INTERFACE I_RpcApi

METHOD CyclicCall
VAR_INPUT
END_VAR
END_METHOD

METHOD RegisterAsynchronousRpcHandlersWith
VAR_INPUT
	Host : I_HostAsynchronousRpcHandlers;
END_VAR
END_METHOD

METHOD RegisterSynchronousRpcHandlersWith
VAR_INPUT
	Host : I_HostSynchronousRpcHandlers;
END_VAR
END_METHOD

END_INTERFACE

(* stored: Version 1.1.0.1, ProductVersion 3.1.4024.12
   Itf I_RpcApi: Id {80fab5d3-ab3c-4589-b1a4-d073091048f6}
   Method CyclicCall: Id {769d4a7e-c9b4-43ef-a71c-993bc6ad988f}
   Method RegisterAsynchronousRpcHandlersWith: Id {8fc48272-b4eb-4ab8-91a9-2766e712e51a}
   Method RegisterSynchronousRpcHandlersWith: Id {19b9dd6b-15e2-4859-9d73-6ffb7cf6f19c} *)
